// TwinCAT 3 PLC project CASE_Anwendung
// ProgramVersion: 3.1.4023.0
// libraries:
//   Tc2_Standard, * (Beckhoff Automation GmbH)
//   Tc2_System, * (Beckhoff Automation GmbH)
//   Tc3_Module, * (Beckhoff Automation GmbH)
// project tree:
//   / PlcTask.TcTTO
//   POUs/ MAIN.TcPOU
//   POUs/Zustandsautomat/DUTs/ States.TcDUT
//   POUs/Zustandsautomat/POU/ Zustandsautomat.TcPOU
// real-time tasks:
//   TASK PlcTask: cycle T#10ms, priority 20, ADS port 350

CONFIGURATION CASE_Anwendung
    RESOURCE PLC ON TwinCAT3
        TASK PlcTask(INTERVAL := T#10ms, PRIORITY := 20);
        PROGRAM MAIN WITH PlcTask : MAIN;
    END_RESOURCE
END_CONFIGURATION

// ---- POUs/Zustandsautomat/DUTs/States.TcDUT
{attribute 'qualified_only'}
{attribute 'strict'}
{attribute 'to_string'}
TYPE States :
(
    Waiting := 0,
    HasCoin,
    ProductEjected,
    CoinEjected
);
END_TYPE

// ---- POUs/MAIN.TcPOU
PROGRAM MAIN
VAR
	Visualisierung		:Visu;
	
	Zustandsautomat1	: Zustandsautomat;
	Panel1				: ST_Panel;
	
	Zustandsautomat2	: Zustandsautomat;
	Panel2				: ST_Panel;
	

END_VAR

Visualisierung();

Zustandsautomat1(
	Panel					:= Panel1,
	ZustandsautomatName 	:= 'Cola Automat',
	AddVisu 					:= Visualisierung);
	
Zustandsautomat2(
	Panel					:= Panel2,
	ZustandsautomatName 	:= 'Fanta Automat',
	AddVisu 					:= Visualisierung);

END_PROGRAM

// ---- POUs/Zustandsautomat/POU/Zustandsautomat.TcPOU
{attribute 'reflection'} 
FUNCTION_BLOCK Zustandsautomat
VAR CONSTANT
	MaxProducts	: UINT := 5;
END_VAR
VAR_INPUT
	Panel				: REFERENCE TO ST_Panel;
	AddVisu				: InterfaceVisu;
	ZustandsautomatName	: STRING(255);

END_VAR
VAR
  State            		: E_States;
  Products         		: UINT := MaxProducts;
  trigButton         	: R_TRIG;
  trigInsertCoin     	: R_TRIG;
  trigTakeProduct    	: R_TRIG;
  trigTakeCoin       	: R_TRIG;


	NeuInit						: BOOL;
//only for VISU
	{attribute 'instance-path'} 
	{attribute 'no_init'} 
	InstanzZustandsautomat		: STRING(255);
 	InstanzNameZustandsautomat	: STRING(255);
END_VAR

Init();
stateMachine();
conditions();

METHOD conditions : BOOL
VAR_INPUT
END_VAR
Panel.NumberOfProducts := Products;
Panel.State := TO_STRING(State);
END_METHOD

METHOD Init : BOOL
VAR_INPUT
END_VAR
VAR
	tempName	: STRING(255);
	nDotFound	: INT;
END_VAR

IF NOT NeuInit THEN
	NeuInit:=TRUE;

	tempName:=InstanzZustandsautomat;
	nDotFound:=FIND(tempName,'.');
	WHILE nDotFound <> 0 DO
		tempName := RIGHT(tempName, LEN(tempName)-nDotFound);
		nDotFound := Tc2_Standard.FIND(tempName, '.');
	END_WHILE

	InstanzNameZustandsautomat := tempName;
	Panel.InstanzName:=InstanzNameZustandsautomat;
	
	IF ADR(Panel) <> 0 THEN
		AddVisu.ZustandsautomatAddVisu(	P_Panel:=ADR(Panel),
										Name := ZustandsautomatName);
	END_IF
								
	
END_IF
END_METHOD

METHOD stateMachine : BOOL
VAR_INPUT
END_VAR
trigButton(CLK := Panel.Button);
trigInsertCoin(CLK := Panel.InsertCoin);
trigTakeProduct(CLK := Panel.TakeProduct);
trigTakeCoin(CLK := Panel.TakeCoin);
 
CASE State OF
  E_States.Waiting:
    IF (trigButton.Q) THEN
      ; // keep in the state
    END_IF
    IF (trigInsertCoin.Q) THEN
      ADSLOGSTR(ADSLOG_MSGTYPE_HINT, 'Customer has insert a coin.', '');
      State := E_States.HasCoin;
    END_IF
 
  E_States.HasCoin:
    IF (trigButton.Q) THEN
      IF (Products > 0) THEN
        Products := Products - 1;
        ADSLOGSTR(ADSLOG_MSGTYPE_HINT, 'Customer has pressed the button. Output product.', '');
        State := E_States.ProductEjected;
      ELSE
        ADSLOGSTR(ADSLOG_MSGTYPE_HINT, 'Customer has pressed the button. No more products. Return coin.', '');
        State := E_States.CoinEjected;
      END_IF
    END_IF
 
  E_States.ProductEjected:
    IF (trigTakeProduct.Q) THEN
      ADSLOGSTR(ADSLOG_MSGTYPE_HINT, 'Customer has taken the product.', '');
      State := E_States.Waiting;
    END_IF
 
  E_States.CoinEjected:
    IF (trigTakeCoin.Q) THEN
      ADSLOGSTR(ADSLOG_MSGTYPE_HINT, 'Customer has taken the coin.', '');
      State := E_States.Waiting;
    END_IF
 
  ELSE
    ADSLOGSTR(ADSLOG_MSGTYPE_ERROR, 'Invalid state', '');
    State := E_States.Waiting;
END_CASE
END_METHOD

END_FUNCTION_BLOCK
